FUNCTION_BLOCK BookingSystem
VAR_INPUT
	mxEnable: BOOL;
	mxnewBookingReqeust: BOOL;
END_VAR
VAR_OUTPUT
	mxDone:BOOL;
	mxError:BOOL;
END_VAR
VAR
	booking: INT;
END_VAR

VAR_IN_OUT
	mwStationStatus: INT;
END_VAR

IF mxEnable THEN
	CASE booking OF
		0:
		 	IF mxnewBookingReqeust THEN
				booking:=10;
			END_IF
		10:
			IF mwStationStatus =100 THEN
				booking:=20;
			ELSE 
				booking:=1000;
			END_IF
		20:
			mwStationStatus:=200;
			booking:=30;
		30:
			mxDone:=TRUE;
			IF NOT mxnewBookingReqeust THEN
				mxDone:=FALSE;
				booking:=0;
			END_IF
		1000:
			mxError:=TRUE;
			IF NOT mxnewBookingReqeust THEN
				mxDone:=FALSE;
				mxError:=FALSE;
				booking:=0;
			END_IF
	END_CASE
END_IF

END_FUNCTION_BLOCK

(* stored: Version 1.1.0.1, ProductVersion 3.1.4024.10
   POU BookingSystem: Id {c179f68b-ad90-4b28-8ed2-dab7bdc95a48}, SpecialFunc None *)
